FUNCTION_BLOCK CMD_bloc
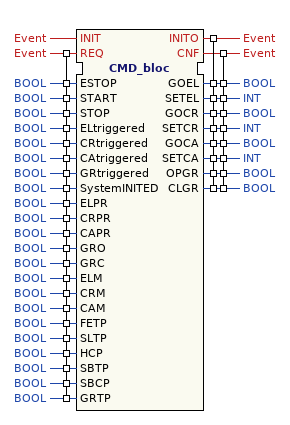
  EVENT_INPUT
    INIT;
    REQ WITH ESTOP, START, STOP, ELtriggered, CRtriggered, CAtriggered, GRtriggered, SystemINITED, ELPR, CRPR, CAPR, GRO, GRC, ELM, CRM, CAM, HCP, SBTP, SBCP, FETP, SLTP, GRTP;
  END_EVENT
  EVENT_OUTPUT
    INITO WITH GOEL, SETEL, GOCA, SETCA, GOCR, SETCR, OPGR, CLGR;
    CNF WITH GOEL, SETEL, GOCA, SETCA, GOCR, SETCR, OPGR, CLGR;
  END_EVENT
  VAR_INPUT
    ESTOP : BOOL;
    START : BOOL;
    STOP : BOOL;
    ELtriggered : BOOL;
    CRtriggered : BOOL;
    CAtriggered : BOOL;
    GRtriggered : BOOL;
    SystemINITED : BOOL;
    ELPR : BOOL;
    CRPR : BOOL;
    CAPR : BOOL;
    GRO : BOOL;
    GRC : BOOL;
    ELM : BOOL;
    CRM : BOOL;
    CAM : BOOL;
    FETP : BOOL;
    SLTP : BOOL;
    HCP : BOOL;
    SBTP : BOOL;
    SBCP : BOOL;
    GRTP : BOOL;
  END_VAR
  VAR_OUTPUT
    GOEL : BOOL;
    SETEL : INT;
    GOCR : BOOL;
    SETCR : INT;
    GOCA : BOOL;
    SETCA : INT;
    OPGR : BOOL;
    CLGR : BOOL;
  END_VAR
  VAR
    i : INT;
  END_VAR
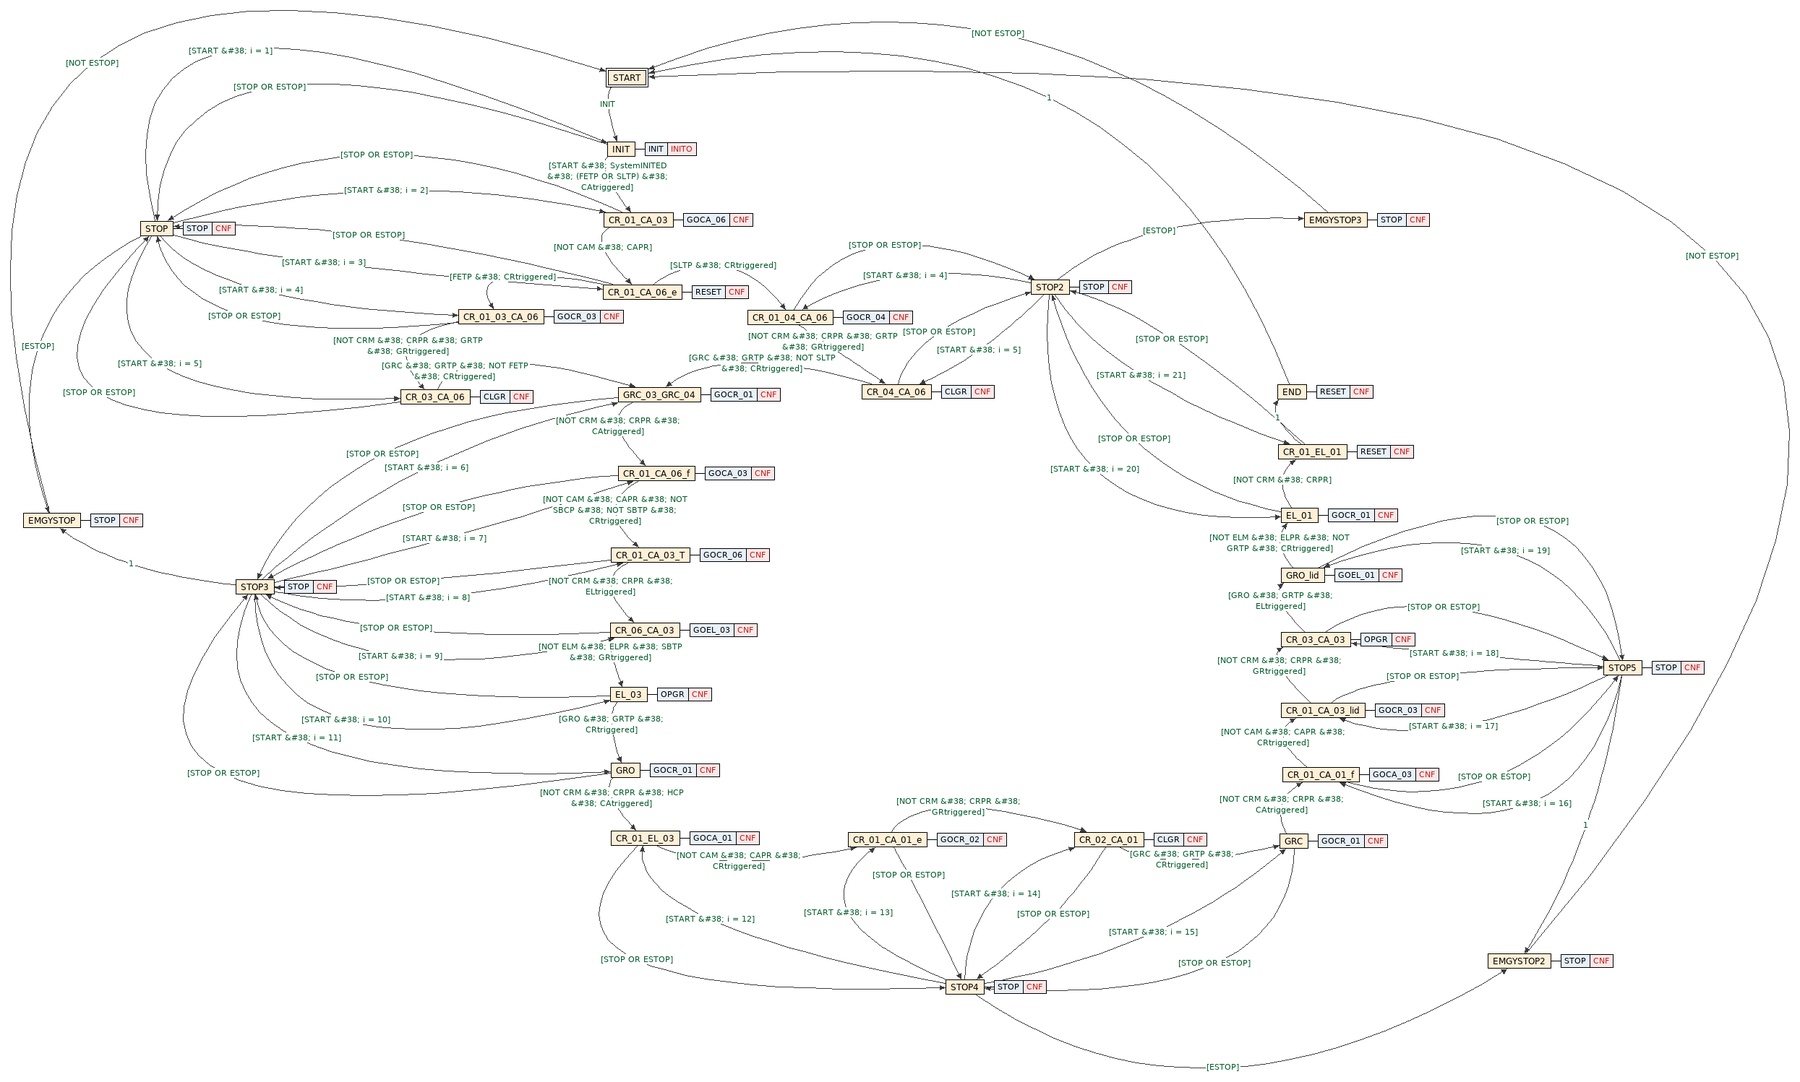
  EC_STATES
    START;
    INIT : INIT -> INITO;
    CR_01_CA_03 : GOCA_06 -> CNF;
    CR_01_03_CA_06 : GOCR_03 -> CNF;
    CR_01_04_CA_06 : GOCR_04 -> CNF;
    GRC_03_GRC_04 : GOCR_01 -> CNF;
    CR_01_CA_06_f : GOCA_03 -> CNF;
    CR_01_CA_03_T : GOCR_06 -> CNF;
    CR_06_CA_03 : GOEL_03 -> CNF;
    EL_03 : OPGR -> CNF;
    GRO : GOCR_01 -> CNF;
    EL_01 : GOCR_01 -> CNF;
    CR_01_EL_03 : GOCA_01 -> CNF;
    END : RESET -> CNF;
    CR_01_CA_01_e : GOCR_02 -> CNF;
    CR_02_CA_01 : CLGR -> CNF;
    GRC : GOCR_01 -> CNF;
    CR_01_CA_01_f : GOCA_03 -> CNF;
    CR_01_CA_03_lid : GOCR_03 -> CNF;
    CR_03_CA_03 : OPGR -> CNF;
    GRO_lid : GOEL_01 -> CNF;
    CR_01_EL_01 : RESET -> CNF;
    CR_01_CA_06_e : RESET -> CNF;
    CR_03_CA_06 : CLGR -> CNF;
    CR_04_CA_06 : CLGR -> CNF;
    STOP : STOP -> CNF;
    STOP2 : STOP -> CNF;
    STOP3 : STOP -> CNF;
    STOP4 : STOP -> CNF;
    STOP5 : STOP -> CNF;
    EMGYSTOP : STOP -> CNF;
    EMGYSTOP2 : STOP -> CNF;
    EMGYSTOP3 : STOP -> CNF;
  END_STATES
  EC_TRANSITIONS
    START TO INIT := INIT;
    CR_01_03_CA_06 TO CR_03_CA_06 := [NOT CRM &#38; CRPR &#38; GRTP &#38; GRtriggered];
    CR_01_04_CA_06 TO CR_04_CA_06 := [NOT CRM &#38; CRPR &#38; GRTP &#38; GRtriggered];
    GRC_03_GRC_04 TO CR_01_CA_06_f := [NOT CRM &#38; CRPR &#38; CAtriggered];
    CR_01_CA_06_f TO CR_01_CA_03_T := [NOT CAM &#38; CAPR &#38; NOT SBCP &#38; NOT SBTP &#38; CRtriggered];
    CR_01_CA_03_T TO CR_06_CA_03 := [NOT CRM &#38; CRPR &#38; ELtriggered];
    CR_06_CA_03 TO EL_03 := [NOT ELM &#38; ELPR &#38; SBTP &#38; GRtriggered];
    EL_03 TO GRO := [GRO &#38; GRTP &#38; CRtriggered];
    GRO TO CR_01_EL_03 := [NOT CRM &#38; CRPR &#38; HCP &#38; CAtriggered];
    CR_01_EL_03 TO CR_01_CA_01_e := [NOT CAM &#38; CAPR &#38; CRtriggered];
    CR_01_CA_01_e TO CR_02_CA_01 := [NOT CRM &#38; CRPR &#38; GRtriggered];
    CR_02_CA_01 TO GRC := [GRC &#38; GRTP &#38; CRtriggered];
    GRC TO CR_01_CA_01_f := [NOT CRM &#38; CRPR &#38; CAtriggered];
    CR_01_CA_01_f TO CR_01_CA_03_lid := [NOT CAM &#38; CAPR &#38; CRtriggered];
    CR_01_CA_03_lid TO CR_03_CA_03 := [NOT CRM &#38; CRPR &#38; GRtriggered];
    CR_03_CA_03 TO GRO_lid := [GRO &#38; GRTP &#38; ELtriggered];
    GRO_lid TO EL_01 := [NOT ELM &#38; ELPR &#38; NOT GRTP &#38; CRtriggered];
    EL_01 TO CR_01_EL_01 := [NOT CRM &#38; CRPR];
    END TO START := 1;
    CR_01_CA_03 TO CR_01_CA_06_e := [NOT CAM &#38; CAPR];
    CR_01_CA_06_e TO CR_01_03_CA_06 := [FETP &#38; CRtriggered];
    CR_01_CA_06_e TO CR_01_04_CA_06 := [SLTP &#38; CRtriggered];
    CR_03_CA_06 TO GRC_03_GRC_04 := [GRC &#38; GRTP &#38; NOT FETP &#38; CRtriggered];
    CR_04_CA_06 TO GRC_03_GRC_04 := [GRC &#38; GRTP &#38; NOT SLTP &#38; CRtriggered];
    INIT TO STOP := [STOP OR ESTOP];
    CR_01_CA_03 TO STOP := [STOP OR ESTOP];
    CR_01_CA_06_e TO STOP := [STOP OR ESTOP];
    CR_01_03_CA_06 TO STOP := [STOP OR ESTOP];
    CR_03_CA_06 TO STOP := [STOP OR ESTOP];
    CR_01_04_CA_06 TO STOP2 := [STOP OR ESTOP];
    CR_04_CA_06 TO STOP2 := [STOP OR ESTOP];
    EL_01 TO STOP2 := [STOP OR ESTOP];
    CR_01_EL_01 TO STOP2 := [STOP OR ESTOP];
    GRC_03_GRC_04 TO STOP3 := [STOP OR ESTOP];
    CR_01_CA_06_f TO STOP3 := [STOP OR ESTOP];
    CR_01_CA_03_T TO STOP3 := [STOP OR ESTOP];
    CR_06_CA_03 TO STOP3 := [STOP OR ESTOP];
    EL_03 TO STOP3 := [STOP OR ESTOP];
    GRO TO STOP3 := [STOP OR ESTOP];
    CR_01_EL_03 TO STOP4 := [STOP OR ESTOP];
    CR_01_CA_01_e TO STOP4 := [STOP OR ESTOP];
    CR_02_CA_01 TO STOP4 := [STOP OR ESTOP];
    GRC TO STOP4 := [STOP OR ESTOP];
    CR_01_CA_01_f TO STOP5 := [STOP OR ESTOP];
    CR_01_CA_03_lid TO STOP5 := [STOP OR ESTOP];
    CR_03_CA_03 TO STOP5 := [STOP OR ESTOP];
    GRO_lid TO STOP5 := [STOP OR ESTOP];
    STOP TO INIT := [START &#38; i = 1];
    STOP TO CR_01_03_CA_06 := [START &#38; i = 4];
    STOP TO CR_03_CA_06 := [START &#38; i = 5];
    STOP TO CR_01_CA_06_e := [START &#38; i = 3];
    STOP TO CR_01_CA_03 := [START &#38; i = 2];
    STOP3 TO GRC_03_GRC_04 := [START &#38; i = 6];
    STOP3 TO CR_01_CA_06_f := [START &#38; i = 7];
    STOP3 TO CR_01_CA_03_T := [START &#38; i = 8];
    STOP3 TO CR_06_CA_03 := [START &#38; i = 9];
    STOP3 TO EL_03 := [START &#38; i = 10];
    STOP3 TO GRO := [START &#38; i = 11];
    STOP4 TO CR_01_EL_03 := [START &#38; i = 12];
    STOP4 TO CR_01_CA_01_e := [START &#38; i = 13];
    STOP4 TO CR_02_CA_01 := [START &#38; i = 14];
    STOP4 TO GRC := [START &#38; i = 15];
    STOP5 TO CR_01_CA_01_f := [START &#38; i = 16];
    STOP5 TO CR_01_CA_03_lid := [START &#38; i = 17];
    STOP5 TO CR_03_CA_03 := [START &#38; i = 18];
    STOP5 TO GRO_lid := [START &#38; i = 19];
    STOP2 TO CR_01_04_CA_06 := [START &#38; i = 4];
    STOP2 TO CR_04_CA_06 := [START &#38; i = 5];
    STOP2 TO CR_01_EL_01 := [START &#38; i = 21];
    STOP2 TO EL_01 := [START &#38; i = 20];
    STOP3 TO EMGYSTOP := 1;
    STOP TO EMGYSTOP := [ESTOP];
    EMGYSTOP TO START := [NOT ESTOP];
    STOP4 TO EMGYSTOP2 := [ESTOP];
    STOP5 TO EMGYSTOP2 := 1;
    STOP2 TO EMGYSTOP3 := [ESTOP];
    EMGYSTOP3 TO START := [NOT ESTOP];
    EMGYSTOP2 TO START := [NOT ESTOP];
    INIT TO CR_01_CA_03 := [START &#38; SystemINITED &#38; (FETP OR SLTP) &#38; CAtriggered];
    CR_01_EL_01 TO END := 1;
  END_TRANSITIONS
  ALGORITHM INIT IN ST:
i := 1;&#38;#10;
  END_ALGORITHM
  ALGORITHM GOCA_06 IN ST:
GOCA := TRUE;&#38;#10;SETCA := 1320;&#38;#10;i := i + 1;&#38;#10;GOEL := FALSE;&#38;#10;GOCR := FALSE;&#38;#10;
  END_ALGORITHM
  ALGORITHM GOCR_03 IN ST:
GOCR := TRUE;&#38;#10;SETCR := 54;&#38;#10;GOCA := FALSE;&#38;#10;GOEL := FALSE;&#38;#10;i := i + 1;&#38;#10;
  END_ALGORITHM
  ALGORITHM GOCR_04 IN ST:
GOCR := TRUE;&#38;#10;SETCR := 81;&#38;#10;GOEL := FALSE;&#38;#10;GOCA := FALSE;&#38;#10;i := i + 1;&#38;#10;
  END_ALGORITHM
  ALGORITHM CLGR IN ST:
CLGR := TRUE;&#38;#10;OPGR := FALSE;&#38;#10;GOCR := FALSE;&#38;#10;GOEL := FALSE;&#38;#10;GOCA := FALSE;&#38;#10;i := i + 1;&#38;#10;
  END_ALGORITHM
  ALGORITHM GOCR_01 IN ST:
GOCR := TRUE;&#38;#10;SETCR := -2;&#38;#10;GOCA := FALSE;&#38;#10;GOEL := FALSE;&#38;#10;FETP := FALSE;&#38;#10;SLTP := FALSE;&#38;#10;i := i + 1;&#38;#10;
  END_ALGORITHM
  ALGORITHM GOCA_03 IN ST:
GOCA := TRUE;&#38;#10;SETCA := 538;&#38;#10;GOEL := FALSE;&#38;#10;GOCR := FALSE;&#38;#10;i := i + 1;&#38;#10;
  END_ALGORITHM
  ALGORITHM GOCR_06 IN ST:
GOCR := TRUE;&#38;#10;SETCR := 261;&#38;#10;GOCA := FALSE;&#38;#10;GOEL := FALSE;&#38;#10;i := i + 1;&#38;#10;
  END_ALGORITHM
  ALGORITHM GOEL_03 IN ST:
GOEL := TRUE;&#38;#10;SETEL := 274;&#38;#10;GOCA := FALSE;&#38;#10;GOCR := FALSE;&#38;#10;i := i + 1;&#38;#10;
  END_ALGORITHM
  ALGORITHM OPGR IN ST:
CLGR := FALSE;&#38;#10;OPGR := TRUE;&#38;#10;GOCR := FALSE;&#38;#10;GOEL := FALSE;&#38;#10;GOCA := FALSE;&#38;#10;i := i + 1;&#38;#10;
  END_ALGORITHM
  ALGORITHM GOCA_01 IN ST:
GOCA := TRUE;&#38;#10;SETCA := 10;&#38;#10;GOEL := FALSE;&#38;#10;GOCR := FALSE;&#38;#10;i := i + 1;&#38;#10;
  END_ALGORITHM
  ALGORITHM GOCR_02 IN ST:
GOCR := TRUE;&#38;#10;SETCR := 41;&#38;#10;GOCA := FALSE;&#38;#10;GOEL := FALSE;&#38;#10;i := i + 1;&#38;#10;
  END_ALGORITHM
  ALGORITHM GOCR_XX IN ST:
GOCR := TRUE;&#38;#10;SETCR := 0;&#38;#10;GOCA := FALSE;&#38;#10;GOEL := FALSE;&#38;#10;
  END_ALGORITHM
  ALGORITHM GOEL_01 IN ST:
GOEL := TRUE;&#38;#10;SETEL := -2;&#38;#10;GOCA := FALSE;&#38;#10;GOCR := FALSE;&#38;#10;i := i + 1;&#38;#10;
  END_ALGORITHM
  ALGORITHM RESET IN ST:
GOCA := FALSE;&#38;#10;GOCR := FALSE;&#38;#10;GOEL := FALSE;&#38;#10;OPGR := FALSE;&#38;#10;CLGR := FALSE;&#38;#10;i := i + 1;&#38;#10;
  END_ALGORITHM
  ALGORITHM STOP IN ST:
GOCA := FALSE;&#38;#10;GOCR := FALSE;&#38;#10;GOEL := FALSE;&#38;#10;OPGR := FALSE;&#38;#10;CLGR := FALSE;&#38;#10;
  END_ALGORITHM
END_FUNCTION_BLOCK
